{attribute 'enable_dynamic_creation'}
FUNCTION_BLOCK ULogger
VAR_INPUT
	bEnable : BOOL;
	bReset : BOOL;
	nBufferSizeSet : UDINT;
	bEnableEventLogger : BOOL;
	bEnableFileLogger : BOOL;
	eSplitLogFileMode : E_LogFileSplitMode := E_LogFileSplitMode.eSplitByDay;
	sLogFilePath : T_MaxString := 'C:\';
	tAutoSave : TIME := T#3M;
END_VAR
VAR_OUTPUT
END_VAR
VAR
	pBufferUsing : POINTER TO BYTE;
	pBufferSaving : POINTER TO BYTE;
	nBufferTotalSize : UDINT;
	nBufferUsedSize : UDINT;
	nBufferSaveSize : UDINT;
	tStartUse : TIME;
	
	bWriteFileRequest : BOOL;
	
	stepWriteFile : INT;
	hFile : UINT;
	fbFileOpen : FB_FileOpen;
	fbFileWrite : FB_FileWrite;
	fbFileClose : FB_FileClose;
	
	
	sFilePathName : T_MaxString;
	
	bError : BOOL;
	
	tonAutoSave : TON;
	tCycleTime : UDINT;
	tPassedTime : UDINT;
	ttimesave: UDINT;
	ttimesavelmt : UDINT;
END_VAR


AutoSave();

CASE stepWriteFile OF
	0:
	IF bWriteFileRequest AND NOT bError THEN
		stepWriteFile := 10;
	ELSIF bError AND bReset THEN
		fbFileOpen(bExecute:= FALSE);
		fbFileWrite(bExecute:= FALSE);
		fbFileClose(bExecute:= FALSE);
		bError := FALSE;
		IF hFile <> 0 THEN
			stepWriteFile := 30;
		END_IF
	END_IF
	10:
	sFilePathName := HandelLogFilePath(SplitLogFileMode:= eSplitLogFileMode, LogFilePath:= sLogFilePath);

	fbFileOpen(sPathName:= sFilePathName, 
		nMode:= FOPEN_MODEAPPEND OR FOPEN_MODETEXT OR FOPEN_MODEPLUS, 
		bExecute:= TRUE);
	IF NOT fbFileOpen.bBusy THEN
		IF NOT fbFileOpen.bError THEN
			hFile := fbFileOpen.hFile;
			stepWriteFile := 20;
		ELSE
			stepWriteFile := 0;
			bError := TRUE;
		END_IF
		fbFileOpen(bExecute:= FALSE);
	END_IF
	20:
	fbFileWrite(
		hFile:= hFile, 
		pWriteBuff:= pBufferSaving, 
		cbWriteLen:= nBufferSaveSize, 
		bExecute:= TRUE);
	IF NOT fbFileWrite.bBusy THEN
		IF NOT fbFileWrite.bError THEN
			stepWriteFile := 30;
		ELSE
			stepWriteFile := 0;
			bError := TRUE;
		END_IF
		fbFileWrite(bExecute:= FALSE);
	END_IF
	30:
	fbFileClose(
		hFile:= hfile, 
		bExecute:= TRUE);
	IF NOT fbFileClose.bBusy THEN
		IF NOT fbFileClose.bError THEN
			hFile := 0;
			stepWriteFile := 0;
			bWriteFileRequest := FALSE;
		ELSE
			hFile := 0;
			bError := TRUE;
			stepWriteFile := 0;
		END_IF
		fbFileClose(bExecute:= FALSE);
	END_IF
END_CASE

METHOD AutoSave : BOOL
VAR_INPUT
END_VAR
IF tCycleTime = 0 THEN
	tCycleTime := _TaskInfo[GETCURTASKINDEXEX()].CycleTime / 10_000;
END_IF
IF nBufferUsedSize > 0 THEN
	tPassedTime := tPassedTime + tCycleTime;
END_IF

ttimesave := TIME_TO_UDINT(tAutoSave);
ttimesavelmt := LIMIT(60_000, ttimesave, 9999_000);
IF tPassedTime >= ttimesavelmt THEN
	SaveBufferNow();
	tPassedTime := 0;
END_IF
END_METHOD

METHOD CreateBuffer : BOOL
VAR_INPUT
END_VAR
VAR
	pTemp : POINTER TO BYTE;
END_VAR
IF nBufferSizeSet = 0 THEN
	RETURN;
END_IF
IF nBufferSizeSet > nBufferTotalSize THEN
	(* 创建使用中缓冲区 *)
	pTemp := __NEW(BYTE, nBufferSizeSet);
	IF pBufferUsing <>0 THEN
		MEMCPY(destAddr:= pTemp, srcAddr:= pBufferUsing, n:= nBufferTotalSize);
		__DELETE(pBufferUsing);
	END_IF
	pBufferUsing := pTemp;
	
	
	(* 创建保存中缓冲区 *)
	pTemp := __NEW(BYTE, nBufferSizeSet);
	IF pBufferSaving <> 0 THEN
		MEMCPY(destAddr:= pTemp, srcAddr:= pBufferSaving, n:= nBufferTotalSize);
		__DELETE(pBufferSaving);
	END_IF
	pBufferSaving := pTemp;
	
	nBufferTotalSize := nBufferSizeSet;
	CreateBuffer := TRUE;
END_IF
END_METHOD

METHOD FB_exit : BOOL
VAR_INPUT
	bInCopyCode : BOOL; // if TRUE, the exit method is called for exiting an instance that is copied afterwards (online change).
END_VAR

VAR
	pBuffer1: INT;
END_VAR
IF NOT bInCopyCode THEN
	IF pBufferUsing <> 0 THEN
		__DELETE(pBufferUsing);
	END_IF
	IF pBufferSaving <> 0 THEN
		__DELETE(pBufferSaving);
	END_IF
	
END_IF
END_METHOD

METHOD HandelLogFilePath : T_MaxString
VAR_INPUT
	SplitLogFileMode : E_LogFileSplitMode;
	LogFilePath : T_MaxString;
END_VAR

VAR
	timestr: DCTIMESTRUCT;
END_VAR
IF SplitLogFileMode = E_LogFileSplitMode.eDontSplit THEN
	HandelLogFilePath := CONCAT(LogFilePath, 'Log.log');
ELSIF eSplitLogFileMode = E_LogFileSplitMode.eSplitByDay THEN
	HandelLogFilePath := CONCAT(LogFilePath, LEFT(STR:= DCTIME64_TO_STRING(F_GetCurDcTaskTime64()), SIZE:= 10));
	HandelLogFilePath := CONCAT(HandelLogFilePath, '.log');
ELSIF eSplitLogFileMode = E_LogFileSplitMode.eSplitByHour THEN
	HandelLogFilePath := CONCAT(LogFilePath, LEFT(STR:= DCTIME64_TO_STRING(F_GetCurDcTaskTime64()), SIZE:= 13));
	HandelLogFilePath := CONCAT(HandelLogFilePath, '.log');
END_IF
END_METHOD

METHOD SaveBufferNow : BOOL
VAR_INPUT
END_VAR
MEMCPY(destAddr:= pBufferSaving, srcAddr:= pBufferUsing, n:= nBufferTotalSize);
nBufferSaveSize := nBufferUsedSize;
nBufferUsedSize := 0;
bWriteFileRequest := TRUE;
END_METHOD

METHOD WriteData : BOOL
VAR_INPUT
	pData : POINTER TO BYTE;
	nSize : UDINT;
END_VAR
IF pData = 0 OR nSize = 0 THEN
	RETURN;
END_IF
IF nBufferSizeSet > nBufferTotalSize THEN
	IF NOT CreateBuffer() THEN
		RETURN;
	END_IF
END_IF
IF nBufferUsedSize = 0 THEN
	tStartUse := TIME();
	IF nSize > nBufferTotalSize THEN
		RETURN;
	END_IF
END_IF
IF nBufferUsedSize + nSize > nBufferTotalSize THEN
	SaveBufferNow();
END_IF

MEMCPY(destAddr:= pBufferUsing + nBufferUsedSize, srcAddr:= pData, n:= nSize);
tPassedTime := 0;
nBufferUsedSize := nBufferUsedSize + nSize;
WriteData := TRUE;
END_METHOD

METHOD WriteLog : BOOL
VAR_INPUT
	LogStr : T_MaxString;
END_VAR
VAR
	Tempstr : STRING;
END_VAR
Tempstr := CONCAT(Tempstr, LEFT(STR:= DCTIME64_TO_STRING(in:= F_GetActualDcTime64()), SIZE:= 27));
Tempstr := CONCAT(Tempstr, ' : ');
Tempstr := CONCAT(Tempstr, LogStr);
Tempstr := CONCAT(Tempstr, '$R');
WriteData(pData:= ADR(Tempstr), nSize:= INT_TO_UDINT(LEN(Tempstr)));
END_METHOD

END_FUNCTION_BLOCK

(* stored: Version 1.1.0.1, ProductVersion 3.1.4024.12
   POU ULogger: Id {f38daff4-e0af-47c8-a4e6-8b569aef59f6}, SpecialFunc None
   Method AutoSave: Id {9ddd61cd-6f56-444e-bdbe-9ef848930c79}
   Method CreateBuffer: Id {74a18b17-aeeb-4579-a67a-2145084862d4}
   Method FB_exit: Id {3c4586a3-7b8a-40c0-8b53-1f075ab3a1f7}
   Method HandelLogFilePath: Id {1deeb122-daa2-45eb-9825-49b2492d5e31}
   Method SaveBufferNow: Id {626f9c74-1002-4dde-bcd7-3e3bb3838e50}
   Method WriteData: Id {26a163d3-4040-4ae5-bf8d-6104fcb7b765}
   Method WriteLog: Id {59fcd53a-573d-409f-b945-e891acadb996} *)
